{attribute 'GeneratedUsingTerminal: EP6224-0042-0016'}
{attribute addProperty BoxType "EP6224-0042-0016"}
{attribute addProperty Id "DI_X01_Pin2AT %I*BOOL1DI_X01_Pin4AT %I*BOOL1DI_X02_Pin2AT %I*BOOL1DI_X02_Pin4AT %I*BOOL1DI_X05_Pin2AT %I*BOOL1DI_X05_Pin4AT %I*BOOL1DI_X06_Pin2AT %I*BOOL1DI_X06_Pin4AT %I*BOOL1"}
{attribute addProperty CRC "2269765969"}
{attribute addProperty Size "8"}
TYPE Digital_Inputs_8749E151 EXTENDS InputBase_8311D824 :
STRUCT
	{attribute addProperty Name "DI_X01_Pin2"}
	DI_X01_Pin2 AT %I* : BOOL;
	{attribute addProperty Name "DI_X01_Pin4"}
	DI_X01_Pin4 AT %I* : BOOL;
	{attribute addProperty Name "DI_X02_Pin2"}
	DI_X02_Pin2 AT %I* : BOOL;
	{attribute addProperty Name "DI_X02_Pin4"}
	DI_X02_Pin4 AT %I* : BOOL;
	{attribute addProperty Name "DI_X05_Pin2"}
	DI_X05_Pin2 AT %I* : BOOL;
	{attribute addProperty Name "DI_X05_Pin4"}
	DI_X05_Pin4 AT %I* : BOOL;
	{attribute addProperty Name "DI_X06_Pin2"}
	DI_X06_Pin2 AT %I* : BOOL;
	{attribute addProperty Name "DI_X06_Pin4"}
	DI_X06_Pin4 AT %I* : BOOL;
END_STRUCT
END_TYPE

(* stored: Version 1.2.0.0, ProductVersion 3.1.4024.9
   DUT Digital_Inputs_8749E151: Id {5007bc9c-827c-44b1-9d6a-ef1f51be0fcd} *)
